// Implement this with I_List to allow a list to be ready only. 
INTERFACE I_Read_Only_List EXTENDS I_Collection

(* DOES NOTHING *)
METHOD Clear
END_METHOD

(* Checks if item is contained in list *)
METHOD Contains : BOOL
VAR_INPUT
	Item : ANY; // Item to find in list
END_VAR
END_METHOD

// Find the location of an item in list.
METHOD Find : I_Read_Only_List
VAR_INPUT
	Item 	: ANY; // Item to find in list
END_VAR
VAR_OUTPUT
	nIndex	: DINT; //Location of item in list 
	bSuccess : BOOL;
END_VAR
END_METHOD

// Gets item from list at specified location without removing it
METHOD Get : I_Read_Only_List
VAR_INPUT
	Return_Item 	: ANY;  // Variable to store returned item
	nIndex 			: DINT; // Location of item
END_VAR
VAR_OUTPUT
	bSuccess : BOOL;
END_VAR
END_METHOD

// Gets item at the front of the list 
METHOD Get_First : I_Read_Only_List
VAR_INPUT
	Return_Item 	: ANY; // Variable to store returned item
END_VAR
VAR_OUTPUT
	bSuccess : BOOL;
END_VAR
END_METHOD

// Gets item at the back of the list 
METHOD Get_Last : I_Read_Only_List
VAR_INPUT
	Return_Item 	: ANY; // Variable to store returned item
END_VAR
VAR_OUTPUT
	bSuccess : BOOL;
END_VAR
END_METHOD

// Returns item as a string, if type to string conversion is supported
METHOD Get_Value_As_String : I_Read_Only_List
VAR_INPUT
	nIndex	: DINT; // Location of item
END_VAR
VAR_OUTPUT
	sItem 	: T_MaxString; // Variable to store returned item
END_VAR
END_METHOD

END_INTERFACE

(* stored: Version 1.1.0.1, ProductVersion 3.1.4024.4
   Itf I_Read_Only_List: Id {2e176e88-c8c5-4847-a1a0-926cf4a92d8d}
   Method Clear: Id {d6995547-57bb-41e7-b8df-fd85f28ecf40}
   Method Contains: Id {8ebb7b9e-4f7b-4cf9-95ea-fc9bd2c187bf}
   Method Find: Id {2f381670-db4f-4ba9-af49-c5db42a5b23e}
   Method Get: Id {d8420af4-ba32-43c3-a53c-e5f508ab733e}
   Method Get_First: Id {6d9e954d-96c6-44c3-a96d-67dfcca65742}
   Method Get_Last: Id {b6ae5e60-f208-437b-9265-4d8e9bf2605e}
   Method Get_Value_As_String: Id {dc3192ff-93fa-4c95-a02b-7ef1166b05a6} *)
